TYPE sJobState :
STRUCT
	boWorkpieceLoaded: BOOL;
	boTransportWorkpiece: BOOL;
	boJobAccepted: BOOL;
	boWaitForRfidOut: BOOL;
	boWaitForRfidIn: BOOL;
	boWorkpiecePlaced: BOOL;
END_STRUCT
END_TYPE

(* stored: Version 1.1.0.1, ProductVersion 3.1.4026.13
   DUT sJobState: Id {acd88359-ba24-42f4-b9f6-d1188ad2f02d} *)
